// TIA Portal V20 export
TYPE "LBP_typeTMLoad"
TITLE = Tool management / Gestion des outils
// User data type for block LBP_TMLoad [DB71] / Type de données utilisateur pour bloc LBP_TMLoad [DB71]
   STRUCT
      IFNo : Array[1..16] of Bool;   // Interface [number] active / Interface [numéro] active
      Quit : Array[1..16] of Bool;   // Perform Quit-End / Effectuer Quit-End
      TIF : Array[1..16] of Struct
         Loading : Bool;   // Loading the tool / Outil en cours de chargement
         Unloading : Bool;   // Unloading the tool / Outil en cours de déchargement
         Reloading : Bool;   // Relocating the tool / Repositionnement de l'outil
         Positioning : Bool;   // Positioning the magazine / Magasin en cours de positionnement
         PosbyProgram : Bool;   // Initiation by CNC program / Initiation par programme CNC
         PositioningMT : Bool;   // Positioning multitool / Multitool en cours de positionnement
         f0_6 : Bool;   // Reserved / Réservé
         f0_7 : Bool;   // Reserved / Réservé
         PerfStatusError : Bool;   // Negative acknowledge / Acquittement négatif
         n1_1 : Bool;   // Reserved / Réservé
         n1_2 : Bool;   // Reserved / Réservé
         n1_3 : Bool;   // Reserved / Réservé
         n1_4 : Bool;   // Reserved / Réservé
         n1_5 : Bool;   // Reserved / Réservé
         n1_6 : Bool;   // Reserved / Réservé
         DataInDB1071 : Bool;   // Multitool data stored in DB1071 / Données Multitool enregistrées dans DB1071
         Channel : Byte;   // Assigned channel / Canal affecté
         TMNo : Byte;   // Tool management number / Numéro de gestion des outils
         reserved1 : DInt;   // Reserved / Réservé
         reserved2 : DInt;   // Reserved / Réservé
         reserved3 : DInt;   // Reserved / Réservé
         LoadIdent : Int;   // Identification for loading/unloading station / Identifiant de la station de chargement/déchargement
         LoadNo : Int;   // Number of loading station / Numéro de la station de chargement
         SMag : Int;   // Magazine number (source) for unloading/reloading/pos. / Numéro de magasin (source) pour déchargement/rechargement/pos.
         SLoc : Int;   // Location number (source) for unloading/reloading/pos. / Numéro d'emplacement (source) pour déchargement/rechargement/pos.
         TMag : Int;   // Magazine number (target) for loading/reloading / Numéro de magasin (cible) pour déchargement/rechargement
         TLoc : Int;   // Location number (target) for loading/reloading / Numéro d'emplacement (cible) pour déchargement/rechargement
         WithoutMagMoving : Bool;   // HMI Data: without magazine moving / Données HMI : sans déplacement du magasin
         Res2 : Byte;   // Reserved / Réservé
      END_STRUCT;
   END_STRUCT;
   // // TIF[2].Loading : Loading the tool / Outil en cours de chargement
   // // TIF[3].Loading : Loading the tool / Outil en cours de chargement
   // // TIF[4].Loading : Loading the tool / Outil en cours de chargement
   // // TIF[5].Loading : Loading the tool / Outil en cours de chargement
   // // TIF[6].Loading : Loading the tool / Outil en cours de chargement
   // // TIF[7].Loading : Loading the tool / Outil en cours de chargement
   // // TIF[8].Loading : Loading the tool / Outil en cours de chargement
   // // TIF[9].Loading : Loading the tool / Outil en cours de chargement
   // // TIF[10].Loading : Loading the tool / Outil en cours de chargement
   // // TIF[11].Loading : Loading the tool / Outil en cours de chargement
   // // TIF[12].Loading : Loading the tool / Outil en cours de chargement
   // // TIF[13].Loading : Loading the tool / Outil en cours de chargement
   // // TIF[14].Loading : Loading the tool / Outil en cours de chargement
   // // TIF[15].Loading : Loading the tool / Outil en cours de chargement
   // // TIF[16].Loading : Loading the tool / Outil en cours de chargement
   // // TIF[2].Unloading : Unloading the tool / Outil en cours de déchargement
   // // TIF[3].Unloading : Unloading the tool / Outil en cours de déchargement
   // // TIF[4].Unloading : Unloading the tool / Outil en cours de déchargement
   // // TIF[5].Unloading : Unloading the tool / Outil en cours de déchargement
   // // TIF[6].Unloading : Unloading the tool / Outil en cours de déchargement
   // // TIF[7].Unloading : Unloading the tool / Outil en cours de déchargement
   // // TIF[8].Unloading : Unloading the tool / Outil en cours de déchargement
   // // TIF[9].Unloading : Unloading the tool / Outil en cours de déchargement
   // // TIF[10].Unloading : Unloading the tool / Outil en cours de déchargement
   // // TIF[11].Unloading : Unloading the tool / Outil en cours de déchargement
   // // TIF[12].Unloading : Unloading the tool / Outil en cours de déchargement
   // // TIF[13].Unloading : Unloading the tool / Outil en cours de déchargement
   // // TIF[14].Unloading : Unloading the tool / Outil en cours de déchargement
   // // TIF[15].Unloading : Unloading the tool / Outil en cours de déchargement
   // // TIF[16].Unloading : Unloading the tool / Outil en cours de déchargement
   // // TIF[2].Reloading : Relocating the tool / Repositionnement de l'outil
   // // TIF[3].Reloading : Relocating the tool / Repositionnement de l'outil
   // // TIF[4].Reloading : Relocating the tool / Repositionnement de l'outil
   // // TIF[5].Reloading : Relocating the tool / Repositionnement de l'outil
   // // TIF[6].Reloading : Relocating the tool / Repositionnement de l'outil
   // // TIF[7].Reloading : Relocating the tool / Repositionnement de l'outil
   // // TIF[8].Reloading : Relocating the tool / Repositionnement de l'outil
   // // TIF[9].Reloading : Relocating the tool / Repositionnement de l'outil
   // // TIF[10].Reloading : Relocating the tool / Repositionnement de l'outil
   // // TIF[11].Reloading : Relocating the tool / Repositionnement de l'outil
   // // TIF[12].Reloading : Relocating the tool / Repositionnement de l'outil
   // // TIF[13].Reloading : Relocating the tool / Repositionnement de l'outil
   // // TIF[14].Reloading : Relocating the tool / Repositionnement de l'outil
   // // TIF[15].Reloading : Relocating the tool / Repositionnement de l'outil
   // // TIF[16].Reloading : Relocating the tool / Repositionnement de l'outil
   // // TIF[2].Positioning : Positioning the magazine / Magasin en cours de positionnement
   // // TIF[3].Positioning : Positioning the magazine / Magasin en cours de positionnement
   // // TIF[4].Positioning : Positioning the magazine / Magasin en cours de positionnement
   // // TIF[5].Positioning : Positioning the magazine / Magasin en cours de positionnement
   // // TIF[6].Positioning : Positioning the magazine / Magasin en cours de positionnement
   // // TIF[7].Positioning : Positioning the magazine / Magasin en cours de positionnement
   // // TIF[8].Positioning : Positioning the magazine / Magasin en cours de positionnement
   // // TIF[9].Positioning : Positioning the magazine / Magasin en cours de positionnement
   // // TIF[10].Positioning : Positioning the magazine / Magasin en cours de positionnement
   // // TIF[11].Positioning : Positioning the magazine / Magasin en cours de positionnement
   // // TIF[12].Positioning : Positioning the magazine / Magasin en cours de positionnement
   // // TIF[13].Positioning : Positioning the magazine / Magasin en cours de positionnement
   // // TIF[14].Positioning : Positioning the magazine / Magasin en cours de positionnement
   // // TIF[15].Positioning : Positioning the magazine / Magasin en cours de positionnement
   // // TIF[16].Positioning : Positioning the magazine / Magasin en cours de positionnement
   // // TIF[2].PosbyProgram : Initiation by CNC program / Initiation par programme CNC
   // // TIF[3].PosbyProgram : Initiation by CNC program / Initiation par programme CNC
   // // TIF[4].PosbyProgram : Initiation by CNC program / Initiation par programme CNC
   // // TIF[5].PosbyProgram : Initiation by CNC program / Initiation par programme CNC
   // // TIF[6].PosbyProgram : Initiation by CNC program / Initiation par programme CNC
   // // TIF[7].PosbyProgram : Initiation by CNC program / Initiation par programme CNC
   // // TIF[8].PosbyProgram : Initiation by CNC program / Initiation par programme CNC
   // // TIF[9].PosbyProgram : Initiation by CNC program / Initiation par programme CNC
   // // TIF[10].PosbyProgram : Initiation by CNC program / Initiation par programme CNC
   // // TIF[11].PosbyProgram : Initiation by CNC program / Initiation par programme CNC
   // // TIF[12].PosbyProgram : Initiation by CNC program / Initiation par programme CNC
   // // TIF[13].PosbyProgram : Initiation by CNC program / Initiation par programme CNC
   // // TIF[14].PosbyProgram : Initiation by CNC program / Initiation par programme CNC
   // // TIF[15].PosbyProgram : Initiation by CNC program / Initiation par programme CNC
   // // TIF[16].PosbyProgram : Initiation by CNC program / Initiation par programme CNC
   // // TIF[2].PositioningMT : Positioning multitool / Multitool en cours de positionnement
   // // TIF[3].PositioningMT : Positioning multitool / Multitool en cours de positionnement
   // // TIF[4].PositioningMT : Positioning multitool / Multitool en cours de positionnement
   // // TIF[5].PositioningMT : Positioning multitool / Multitool en cours de positionnement
   // // TIF[6].PositioningMT : Positioning multitool / Multitool en cours de positionnement
   // // TIF[7].PositioningMT : Positioning multitool / Multitool en cours de positionnement
   // // TIF[8].PositioningMT : Positioning multitool / Multitool en cours de positionnement
   // // TIF[9].PositioningMT : Positioning multitool / Multitool en cours de positionnement
   // // TIF[10].PositioningMT : Positioning multitool / Multitool en cours de positionnement
   // // TIF[11].PositioningMT : Positioning multitool / Multitool en cours de positionnement
   // // TIF[12].PositioningMT : Positioning multitool / Multitool en cours de positionnement
   // // TIF[13].PositioningMT : Positioning multitool / Multitool en cours de positionnement
   // // TIF[14].PositioningMT : Positioning multitool / Multitool en cours de positionnement
   // // TIF[15].PositioningMT : Positioning multitool / Multitool en cours de positionnement
   // // TIF[16].PositioningMT : Positioning multitool / Multitool en cours de positionnement
   // // TIF[2].f0_6 : Reserved / Réservé
   // // TIF[3].f0_6 : Reserved / Réservé
   // // TIF[4].f0_6 : Reserved / Réservé
   // // TIF[5].f0_6 : Reserved / Réservé
   // // TIF[6].f0_6 : Reserved / Réservé
   // // TIF[7].f0_6 : Reserved / Réservé
   // // TIF[8].f0_6 : Reserved / Réservé
   // // TIF[9].f0_6 : Reserved / Réservé
   // // TIF[10].f0_6 : Reserved / Réservé
   // // TIF[11].f0_6 : Reserved / Réservé
   // // TIF[12].f0_6 : Reserved / Réservé
   // // TIF[13].f0_6 : Reserved / Réservé
   // // TIF[14].f0_6 : Reserved / Réservé
   // // TIF[15].f0_6 : Reserved / Réservé
   // // TIF[16].f0_6 : Reserved / Réservé
   // // TIF[2].f0_7 : Reserved / Réservé
   // // TIF[3].f0_7 : Reserved / Réservé
   // // TIF[4].f0_7 : Reserved / Réservé
   // // TIF[5].f0_7 : Reserved / Réservé
   // // TIF[6].f0_7 : Reserved / Réservé
   // // TIF[7].f0_7 : Reserved / Réservé
   // // TIF[8].f0_7 : Reserved / Réservé
   // // TIF[9].f0_7 : Reserved / Réservé
   // // TIF[10].f0_7 : Reserved / Réservé
   // // TIF[11].f0_7 : Reserved / Réservé
   // // TIF[12].f0_7 : Reserved / Réservé
   // // TIF[13].f0_7 : Reserved / Réservé
   // // TIF[14].f0_7 : Reserved / Réservé
   // // TIF[15].f0_7 : Reserved / Réservé
   // // TIF[16].f0_7 : Reserved / Réservé
   // // TIF[2].PerfStatusError : Negative acknowledge / Acquittement négatif
   // // TIF[3].PerfStatusError : Negative acknowledge / Acquittement négatif
   // // TIF[4].PerfStatusError : Negative acknowledge / Acquittement négatif
   // // TIF[5].PerfStatusError : Negative acknowledge / Acquittement négatif
   // // TIF[6].PerfStatusError : Negative acknowledge / Acquittement négatif
   // // TIF[7].PerfStatusError : Negative acknowledge / Acquittement négatif
   // // TIF[8].PerfStatusError : Negative acknowledge / Acquittement négatif
   // // TIF[9].PerfStatusError : Negative acknowledge / Acquittement négatif
   // // TIF[10].PerfStatusError : Negative acknowledge / Acquittement négatif
   // // TIF[11].PerfStatusError : Negative acknowledge / Acquittement négatif
   // // TIF[12].PerfStatusError : Negative acknowledge / Acquittement négatif
   // // TIF[13].PerfStatusError : Negative acknowledge / Acquittement négatif
   // // TIF[14].PerfStatusError : Negative acknowledge / Acquittement négatif
   // // TIF[15].PerfStatusError : Negative acknowledge / Acquittement négatif
   // // TIF[16].PerfStatusError : Negative acknowledge / Acquittement négatif
   // // TIF[2].n1_1 : Reserved / Réservé
   // // TIF[3].n1_1 : Reserved / Réservé
   // // TIF[4].n1_1 : Reserved / Réservé
   // // TIF[5].n1_1 : Reserved / Réservé
   // // TIF[6].n1_1 : Reserved / Réservé
   // // TIF[7].n1_1 : Reserved / Réservé
   // // TIF[8].n1_1 : Reserved / Réservé
   // // TIF[9].n1_1 : Reserved / Réservé
   // // TIF[10].n1_1 : Reserved / Réservé
   // // TIF[11].n1_1 : Reserved / Réservé
   // // TIF[12].n1_1 : Reserved / Réservé
   // // TIF[13].n1_1 : Reserved / Réservé
   // // TIF[14].n1_1 : Reserved / Réservé
   // // TIF[15].n1_1 : Reserved / Réservé
   // // TIF[16].n1_1 : Reserved / Réservé
   // // TIF[2].n1_2 : Reserved / Réservé
   // // TIF[3].n1_2 : Reserved / Réservé
   // // TIF[4].n1_2 : Reserved / Réservé
   // // TIF[5].n1_2 : Reserved / Réservé
   // // TIF[6].n1_2 : Reserved / Réservé
   // // TIF[7].n1_2 : Reserved / Réservé
   // // TIF[8].n1_2 : Reserved / Réservé
   // // TIF[9].n1_2 : Reserved / Réservé
   // // TIF[10].n1_2 : Reserved / Réservé
   // // TIF[11].n1_2 : Reserved / Réservé
   // // TIF[12].n1_2 : Reserved / Réservé
   // // TIF[13].n1_2 : Reserved / Réservé
   // // TIF[14].n1_2 : Reserved / Réservé
   // // TIF[15].n1_2 : Reserved / Réservé
   // // TIF[16].n1_2 : Reserved / Réservé
   // // TIF[2].n1_3 : Reserved / Réservé
   // // TIF[3].n1_3 : Reserved / Réservé
   // // TIF[4].n1_3 : Reserved / Réservé
   // // TIF[5].n1_3 : Reserved / Réservé
   // // TIF[6].n1_3 : Reserved / Réservé
   // // TIF[7].n1_3 : Reserved / Réservé
   // // TIF[8].n1_3 : Reserved / Réservé
   // // TIF[9].n1_3 : Reserved / Réservé
   // // TIF[10].n1_3 : Reserved / Réservé
   // // TIF[11].n1_3 : Reserved / Réservé
   // // TIF[12].n1_3 : Reserved / Réservé
   // // TIF[13].n1_3 : Reserved / Réservé
   // // TIF[14].n1_3 : Reserved / Réservé
   // // TIF[15].n1_3 : Reserved / Réservé
   // // TIF[16].n1_3 : Reserved / Réservé
   // // TIF[2].n1_4 : Reserved / Réservé
   // // TIF[3].n1_4 : Reserved / Réservé
   // // TIF[4].n1_4 : Reserved / Réservé
   // // TIF[5].n1_4 : Reserved / Réservé
   // // TIF[6].n1_4 : Reserved / Réservé
   // // TIF[7].n1_4 : Reserved / Réservé
   // // TIF[8].n1_4 : Reserved / Réservé
   // // TIF[9].n1_4 : Reserved / Réservé
   // // TIF[10].n1_4 : Reserved / Réservé
   // // TIF[11].n1_4 : Reserved / Réservé
   // // TIF[12].n1_4 : Reserved / Réservé
   // // TIF[13].n1_4 : Reserved / Réservé
   // // TIF[14].n1_4 : Reserved / Réservé
   // // TIF[15].n1_4 : Reserved / Réservé
   // // TIF[16].n1_4 : Reserved / Réservé
   // // TIF[2].n1_5 : Reserved / Réservé
   // // TIF[3].n1_5 : Reserved / Réservé
   // // TIF[4].n1_5 : Reserved / Réservé
   // // TIF[5].n1_5 : Reserved / Réservé
   // // TIF[6].n1_5 : Reserved / Réservé
   // // TIF[7].n1_5 : Reserved / Réservé
   // // TIF[8].n1_5 : Reserved / Réservé
   // // TIF[9].n1_5 : Reserved / Réservé
   // // TIF[10].n1_5 : Reserved / Réservé
   // // TIF[11].n1_5 : Reserved / Réservé
   // // TIF[12].n1_5 : Reserved / Réservé
   // // TIF[13].n1_5 : Reserved / Réservé
   // // TIF[14].n1_5 : Reserved / Réservé
   // // TIF[15].n1_5 : Reserved / Réservé
   // // TIF[16].n1_5 : Reserved / Réservé
   // // TIF[2].n1_6 : Reserved / Réservé
   // // TIF[3].n1_6 : Reserved / Réservé
   // // TIF[4].n1_6 : Reserved / Réservé
   // // TIF[5].n1_6 : Reserved / Réservé
   // // TIF[6].n1_6 : Reserved / Réservé
   // // TIF[7].n1_6 : Reserved / Réservé
   // // TIF[8].n1_6 : Reserved / Réservé
   // // TIF[9].n1_6 : Reserved / Réservé
   // // TIF[10].n1_6 : Reserved / Réservé
   // // TIF[11].n1_6 : Reserved / Réservé
   // // TIF[12].n1_6 : Reserved / Réservé
   // // TIF[13].n1_6 : Reserved / Réservé
   // // TIF[14].n1_6 : Reserved / Réservé
   // // TIF[15].n1_6 : Reserved / Réservé
   // // TIF[16].n1_6 : Reserved / Réservé
   // // TIF[2].DataInDB1071 : Multitool data stored in DB1071 / Données Multitool enregistrées dans DB1071
   // // TIF[3].DataInDB1071 : Multitool data stored in DB1071 / Données Multitool enregistrées dans DB1071
   // // TIF[4].DataInDB1071 : Multitool data stored in DB1071 / Données Multitool enregistrées dans DB1071
   // // TIF[5].DataInDB1071 : Multitool data stored in DB1071 / Données Multitool enregistrées dans DB1071
   // // TIF[6].DataInDB1071 : Multitool data stored in DB1071 / Données Multitool enregistrées dans DB1071
   // // TIF[7].DataInDB1071 : Multitool data stored in DB1071 / Données Multitool enregistrées dans DB1071
   // // TIF[8].DataInDB1071 : Multitool data stored in DB1071 / Données Multitool enregistrées dans DB1071
   // // TIF[9].DataInDB1071 : Multitool data stored in DB1071 / Données Multitool enregistrées dans DB1071
   // // TIF[10].DataInDB1071 : Multitool data stored in DB1071 / Données Multitool enregistrées dans DB1071
   // // TIF[11].DataInDB1071 : Multitool data stored in DB1071 / Données Multitool enregistrées dans DB1071
   // // TIF[12].DataInDB1071 : Multitool data stored in DB1071 / Données Multitool enregistrées dans DB1071
   // // TIF[13].DataInDB1071 : Multitool data stored in DB1071 / Données Multitool enregistrées dans DB1071
   // // TIF[14].DataInDB1071 : Multitool data stored in DB1071 / Données Multitool enregistrées dans DB1071
   // // TIF[15].DataInDB1071 : Multitool data stored in DB1071 / Données Multitool enregistrées dans DB1071
   // // TIF[16].DataInDB1071 : Multitool data stored in DB1071 / Données Multitool enregistrées dans DB1071
   // // TIF[2].Channel : Assigned channel / Canal affecté
   // // TIF[3].Channel : Assigned channel / Canal affecté
   // // TIF[4].Channel : Assigned channel / Canal affecté
   // // TIF[5].Channel : Assigned channel / Canal affecté
   // // TIF[6].Channel : Assigned channel / Canal affecté
   // // TIF[7].Channel : Assigned channel / Canal affecté
   // // TIF[8].Channel : Assigned channel / Canal affecté
   // // TIF[9].Channel : Assigned channel / Canal affecté
   // // TIF[10].Channel : Assigned channel / Canal affecté
   // // TIF[11].Channel : Assigned channel / Canal affecté
   // // TIF[12].Channel : Assigned channel / Canal affecté
   // // TIF[13].Channel : Assigned channel / Canal affecté
   // // TIF[14].Channel : Assigned channel / Canal affecté
   // // TIF[15].Channel : Assigned channel / Canal affecté
   // // TIF[16].Channel : Assigned channel / Canal affecté
   // // TIF[2].TMNo : Tool management number / Numéro de gestion des outils
   // // TIF[3].TMNo : Tool management number / Numéro de gestion des outils
   // // TIF[4].TMNo : Tool management number / Numéro de gestion des outils
   // // TIF[5].TMNo : Tool management number / Numéro de gestion des outils
   // // TIF[6].TMNo : Tool management number / Numéro de gestion des outils
   // // TIF[7].TMNo : Tool management number / Numéro de gestion des outils
   // // TIF[8].TMNo : Tool management number / Numéro de gestion des outils
   // // TIF[9].TMNo : Tool management number / Numéro de gestion des outils
   // // TIF[10].TMNo : Tool management number / Numéro de gestion des outils
   // // TIF[11].TMNo : Tool management number / Numéro de gestion des outils
   // // TIF[12].TMNo : Tool management number / Numéro de gestion des outils
   // // TIF[13].TMNo : Tool management number / Numéro de gestion des outils
   // // TIF[14].TMNo : Tool management number / Numéro de gestion des outils
   // // TIF[15].TMNo : Tool management number / Numéro de gestion des outils
   // // TIF[16].TMNo : Tool management number / Numéro de gestion des outils
   // // TIF[2].reserved1 : Reserved / Réservé
   // // TIF[3].reserved1 : Reserved / Réservé
   // // TIF[4].reserved1 : Reserved / Réservé
   // // TIF[5].reserved1 : Reserved / Réservé
   // // TIF[6].reserved1 : Reserved / Réservé
   // // TIF[7].reserved1 : Reserved / Réservé
   // // TIF[8].reserved1 : Reserved / Réservé
   // // TIF[9].reserved1 : Reserved / Réservé
   // // TIF[10].reserved1 : Reserved / Réservé
   // // TIF[11].reserved1 : Reserved / Réservé
   // // TIF[12].reserved1 : Reserved / Réservé
   // // TIF[13].reserved1 : Reserved / Réservé
   // // TIF[14].reserved1 : Reserved / Réservé
   // // TIF[15].reserved1 : Reserved / Réservé
   // // TIF[16].reserved1 : Reserved / Réservé
   // // TIF[2].reserved2 : Reserved / Réservé
   // // TIF[3].reserved2 : Reserved / Réservé
   // // TIF[4].reserved2 : Reserved / Réservé
   // // TIF[5].reserved2 : Reserved / Réservé
   // // TIF[6].reserved2 : Reserved / Réservé
   // // TIF[7].reserved2 : Reserved / Réservé
   // // TIF[8].reserved2 : Reserved / Réservé
   // // TIF[9].reserved2 : Reserved / Réservé
   // // TIF[10].reserved2 : Reserved / Réservé
   // // TIF[11].reserved2 : Reserved / Réservé
   // // TIF[12].reserved2 : Reserved / Réservé
   // // TIF[13].reserved2 : Reserved / Réservé
   // // TIF[14].reserved2 : Reserved / Réservé
   // // TIF[15].reserved2 : Reserved / Réservé
   // // TIF[16].reserved2 : Reserved / Réservé
   // // TIF[2].reserved3 : Reserved / Réservé
   // // TIF[3].reserved3 : Reserved / Réservé
   // // TIF[4].reserved3 : Reserved / Réservé
   // // TIF[5].reserved3 : Reserved / Réservé
   // // TIF[6].reserved3 : Reserved / Réservé
   // // TIF[7].reserved3 : Reserved / Réservé
   // // TIF[8].reserved3 : Reserved / Réservé
   // // TIF[9].reserved3 : Reserved / Réservé
   // // TIF[10].reserved3 : Reserved / Réservé
   // // TIF[11].reserved3 : Reserved / Réservé
   // // TIF[12].reserved3 : Reserved / Réservé
   // // TIF[13].reserved3 : Reserved / Réservé
   // // TIF[14].reserved3 : Reserved / Réservé
   // // TIF[15].reserved3 : Reserved / Réservé
   // // TIF[16].reserved3 : Reserved / Réservé
   // // TIF[2].LoadIdent : Identification for loading/unloading station / Identifiant de la station de chargement/déchargement
   // // TIF[3].LoadIdent : Identification for loading/unloading station / Identifiant de la station de chargement/déchargement
   // // TIF[4].LoadIdent : Identification for loading/unloading station / Identifiant de la station de chargement/déchargement
   // // TIF[5].LoadIdent : Identification for loading/unloading station / Identifiant de la station de chargement/déchargement
   // // TIF[6].LoadIdent : Identification for loading/unloading station / Identifiant de la station de chargement/déchargement
   // // TIF[7].LoadIdent : Identification for loading/unloading station / Identifiant de la station de chargement/déchargement
   // // TIF[8].LoadIdent : Identification for loading/unloading station / Identifiant de la station de chargement/déchargement
   // // TIF[9].LoadIdent : Identification for loading/unloading station / Identifiant de la station de chargement/déchargement
   // // TIF[10].LoadIdent : Identification for loading/unloading station / Identifiant de la station de chargement/déchargement
   // // TIF[11].LoadIdent : Identification for loading/unloading station / Identifiant de la station de chargement/déchargement
   // // TIF[12].LoadIdent : Identification for loading/unloading station / Identifiant de la station de chargement/déchargement
   // // TIF[13].LoadIdent : Identification for loading/unloading station / Identifiant de la station de chargement/déchargement
   // // TIF[14].LoadIdent : Identification for loading/unloading station / Identifiant de la station de chargement/déchargement
   // // TIF[15].LoadIdent : Identification for loading/unloading station / Identifiant de la station de chargement/déchargement
   // // TIF[16].LoadIdent : Identification for loading/unloading station / Identifiant de la station de chargement/déchargement
   // // TIF[2].LoadNo : Number of loading station / Numéro de la station de chargement
   // // TIF[3].LoadNo : Number of loading station / Numéro de la station de chargement
   // // TIF[4].LoadNo : Number of loading station / Numéro de la station de chargement
   // // TIF[5].LoadNo : Number of loading station / Numéro de la station de chargement
   // // TIF[6].LoadNo : Number of loading station / Numéro de la station de chargement
   // // TIF[7].LoadNo : Number of loading station / Numéro de la station de chargement
   // // TIF[8].LoadNo : Number of loading station / Numéro de la station de chargement
   // // TIF[9].LoadNo : Number of loading station / Numéro de la station de chargement
   // // TIF[10].LoadNo : Number of loading station / Numéro de la station de chargement
   // // TIF[11].LoadNo : Number of loading station / Numéro de la station de chargement
   // // TIF[12].LoadNo : Number of loading station / Numéro de la station de chargement
   // // TIF[13].LoadNo : Number of loading station / Numéro de la station de chargement
   // // TIF[14].LoadNo : Number of loading station / Numéro de la station de chargement
   // // TIF[15].LoadNo : Number of loading station / Numéro de la station de chargement
   // // TIF[16].LoadNo : Number of loading station / Numéro de la station de chargement
   // // TIF[2].SMag : Magazine number (source) for unloading/reloading/pos. / Numéro de magasin (source) pour déchargement/rechargement/pos.
   // // TIF[3].SMag : Magazine number (source) for unloading/reloading/pos. / Numéro de magasin (source) pour déchargement/rechargement/pos.
   // // TIF[4].SMag : Magazine number (source) for unloading/reloading/pos. / Numéro de magasin (source) pour déchargement/rechargement/pos.
   // // TIF[5].SMag : Magazine number (source) for unloading/reloading/pos. / Numéro de magasin (source) pour déchargement/rechargement/pos.
   // // TIF[6].SMag : Magazine number (source) for unloading/reloading/pos. / Numéro de magasin (source) pour déchargement/rechargement/pos.
   // // TIF[7].SMag : Magazine number (source) for unloading/reloading/pos. / Numéro de magasin (source) pour déchargement/rechargement/pos.
   // // TIF[8].SMag : Magazine number (source) for unloading/reloading/pos. / Numéro de magasin (source) pour déchargement/rechargement/pos.
   // // TIF[9].SMag : Magazine number (source) for unloading/reloading/pos. / Numéro de magasin (source) pour déchargement/rechargement/pos.
   // // TIF[10].SMag : Magazine number (source) for unloading/reloading/pos. / Numéro de magasin (source) pour déchargement/rechargement/pos.
   // // TIF[11].SMag : Magazine number (source) for unloading/reloading/pos. / Numéro de magasin (source) pour déchargement/rechargement/pos.
   // // TIF[12].SMag : Magazine number (source) for unloading/reloading/pos. / Numéro de magasin (source) pour déchargement/rechargement/pos.
   // // TIF[13].SMag : Magazine number (source) for unloading/reloading/pos. / Numéro de magasin (source) pour déchargement/rechargement/pos.
   // // TIF[14].SMag : Magazine number (source) for unloading/reloading/pos. / Numéro de magasin (source) pour déchargement/rechargement/pos.
   // // TIF[15].SMag : Magazine number (source) for unloading/reloading/pos. / Numéro de magasin (source) pour déchargement/rechargement/pos.
   // // TIF[16].SMag : Magazine number (source) for unloading/reloading/pos. / Numéro de magasin (source) pour déchargement/rechargement/pos.
   // // TIF[2].SLoc : Location number (source) for unloading/reloading/pos. / Numéro d'emplacement (source) pour déchargement/rechargement/pos.
   // // TIF[3].SLoc : Location number (source) for unloading/reloading/pos. / Numéro d'emplacement (source) pour déchargement/rechargement/pos.
   // // TIF[4].SLoc : Location number (source) for unloading/reloading/pos. / Numéro d'emplacement (source) pour déchargement/rechargement/pos.
   // // TIF[5].SLoc : Location number (source) for unloading/reloading/pos. / Numéro d'emplacement (source) pour déchargement/rechargement/pos.
   // // TIF[6].SLoc : Location number (source) for unloading/reloading/pos. / Numéro d'emplacement (source) pour déchargement/rechargement/pos.
   // // TIF[7].SLoc : Location number (source) for unloading/reloading/pos. / Numéro d'emplacement (source) pour déchargement/rechargement/pos.
   // // TIF[8].SLoc : Location number (source) for unloading/reloading/pos. / Numéro d'emplacement (source) pour déchargement/rechargement/pos.
   // // TIF[9].SLoc : Location number (source) for unloading/reloading/pos. / Numéro d'emplacement (source) pour déchargement/rechargement/pos.
   // // TIF[10].SLoc : Location number (source) for unloading/reloading/pos. / Numéro d'emplacement (source) pour déchargement/rechargement/pos.
   // // TIF[11].SLoc : Location number (source) for unloading/reloading/pos. / Numéro d'emplacement (source) pour déchargement/rechargement/pos.
   // // TIF[12].SLoc : Location number (source) for unloading/reloading/pos. / Numéro d'emplacement (source) pour déchargement/rechargement/pos.
   // // TIF[13].SLoc : Location number (source) for unloading/reloading/pos. / Numéro d'emplacement (source) pour déchargement/rechargement/pos.
   // // TIF[14].SLoc : Location number (source) for unloading/reloading/pos. / Numéro d'emplacement (source) pour déchargement/rechargement/pos.
   // // TIF[15].SLoc : Location number (source) for unloading/reloading/pos. / Numéro d'emplacement (source) pour déchargement/rechargement/pos.
   // // TIF[16].SLoc : Location number (source) for unloading/reloading/pos. / Numéro d'emplacement (source) pour déchargement/rechargement/pos.
   // // TIF[2].TMag : Magazine number (target) for loading/reloading / Numéro de magasin (cible) pour déchargement/rechargement
   // // TIF[3].TMag : Magazine number (target) for loading/reloading / Numéro de magasin (cible) pour déchargement/rechargement
   // // TIF[4].TMag : Magazine number (target) for loading/reloading / Numéro de magasin (cible) pour déchargement/rechargement
   // // TIF[5].TMag : Magazine number (target) for loading/reloading / Numéro de magasin (cible) pour déchargement/rechargement
   // // TIF[6].TMag : Magazine number (target) for loading/reloading / Numéro de magasin (cible) pour déchargement/rechargement
   // // TIF[7].TMag : Magazine number (target) for loading/reloading / Numéro de magasin (cible) pour déchargement/rechargement
   // // TIF[8].TMag : Magazine number (target) for loading/reloading / Numéro de magasin (cible) pour déchargement/rechargement
   // // TIF[9].TMag : Magazine number (target) for loading/reloading / Numéro de magasin (cible) pour déchargement/rechargement
   // // TIF[10].TMag : Magazine number (target) for loading/reloading / Numéro de magasin (cible) pour déchargement/rechargement
   // // TIF[11].TMag : Magazine number (target) for loading/reloading / Numéro de magasin (cible) pour déchargement/rechargement
   // // TIF[12].TMag : Magazine number (target) for loading/reloading / Numéro de magasin (cible) pour déchargement/rechargement
   // // TIF[13].TMag : Magazine number (target) for loading/reloading / Numéro de magasin (cible) pour déchargement/rechargement
   // // TIF[14].TMag : Magazine number (target) for loading/reloading / Numéro de magasin (cible) pour déchargement/rechargement
   // // TIF[15].TMag : Magazine number (target) for loading/reloading / Numéro de magasin (cible) pour déchargement/rechargement
   // // TIF[16].TMag : Magazine number (target) for loading/reloading / Numéro de magasin (cible) pour déchargement/rechargement
   // // TIF[2].TLoc : Location number (target) for loading/reloading / Numéro d'emplacement (cible) pour déchargement/rechargement
   // // TIF[3].TLoc : Location number (target) for loading/reloading / Numéro d'emplacement (cible) pour déchargement/rechargement
   // // TIF[4].TLoc : Location number (target) for loading/reloading / Numéro d'emplacement (cible) pour déchargement/rechargement
   // // TIF[5].TLoc : Location number (target) for loading/reloading / Numéro d'emplacement (cible) pour déchargement/rechargement
   // // TIF[6].TLoc : Location number (target) for loading/reloading / Numéro d'emplacement (cible) pour déchargement/rechargement
   // // TIF[7].TLoc : Location number (target) for loading/reloading / Numéro d'emplacement (cible) pour déchargement/rechargement
   // // TIF[8].TLoc : Location number (target) for loading/reloading / Numéro d'emplacement (cible) pour déchargement/rechargement
   // // TIF[9].TLoc : Location number (target) for loading/reloading / Numéro d'emplacement (cible) pour déchargement/rechargement
   // // TIF[10].TLoc : Location number (target) for loading/reloading / Numéro d'emplacement (cible) pour déchargement/rechargement
   // // TIF[11].TLoc : Location number (target) for loading/reloading / Numéro d'emplacement (cible) pour déchargement/rechargement
   // // TIF[12].TLoc : Location number (target) for loading/reloading / Numéro d'emplacement (cible) pour déchargement/rechargement
   // // TIF[13].TLoc : Location number (target) for loading/reloading / Numéro d'emplacement (cible) pour déchargement/rechargement
   // // TIF[14].TLoc : Location number (target) for loading/reloading / Numéro d'emplacement (cible) pour déchargement/rechargement
   // // TIF[15].TLoc : Location number (target) for loading/reloading / Numéro d'emplacement (cible) pour déchargement/rechargement
   // // TIF[16].TLoc : Location number (target) for loading/reloading / Numéro d'emplacement (cible) pour déchargement/rechargement
   // // TIF[2].WithoutMagMoving : HMI Data: without magazine moving / Données HMI : sans déplacement du magasin
   // // TIF[3].WithoutMagMoving : HMI Data: without magazine moving / Données HMI : sans déplacement du magasin
   // // TIF[4].WithoutMagMoving : HMI Data: without magazine moving / Données HMI : sans déplacement du magasin
   // // TIF[5].WithoutMagMoving : HMI Data: without magazine moving / Données HMI : sans déplacement du magasin
   // // TIF[6].WithoutMagMoving : HMI Data: without magazine moving / Données HMI : sans déplacement du magasin
   // // TIF[7].WithoutMagMoving : HMI Data: without magazine moving / Données HMI : sans déplacement du magasin
   // // TIF[8].WithoutMagMoving : HMI Data: without magazine moving / Données HMI : sans déplacement du magasin
   // // TIF[9].WithoutMagMoving : HMI Data: without magazine moving / Données HMI : sans déplacement du magasin
   // // TIF[10].WithoutMagMoving : HMI Data: without magazine moving / Données HMI : sans déplacement du magasin
   // // TIF[11].WithoutMagMoving : HMI Data: without magazine moving / Données HMI : sans déplacement du magasin
   // // TIF[12].WithoutMagMoving : HMI Data: without magazine moving / Données HMI : sans déplacement du magasin
   // // TIF[13].WithoutMagMoving : HMI Data: without magazine moving / Données HMI : sans déplacement du magasin
   // // TIF[14].WithoutMagMoving : HMI Data: without magazine moving / Données HMI : sans déplacement du magasin
   // // TIF[15].WithoutMagMoving : HMI Data: without magazine moving / Données HMI : sans déplacement du magasin
   // // TIF[16].WithoutMagMoving : HMI Data: without magazine moving / Données HMI : sans déplacement du magasin
   // // TIF[2].Res2 : Reserved / Réservé
   // // TIF[3].Res2 : Reserved / Réservé
   // // TIF[4].Res2 : Reserved / Réservé
   // // TIF[5].Res2 : Reserved / Réservé
   // // TIF[6].Res2 : Reserved / Réservé
   // // TIF[7].Res2 : Reserved / Réservé
   // // TIF[8].Res2 : Reserved / Réservé
   // // TIF[9].Res2 : Reserved / Réservé
   // // TIF[10].Res2 : Reserved / Réservé
   // // TIF[11].Res2 : Reserved / Réservé
   // // TIF[12].Res2 : Reserved / Réservé
   // // TIF[13].Res2 : Reserved / Réservé
   // // TIF[14].Res2 : Reserved / Réservé
   // // TIF[15].Res2 : Reserved / Réservé
   // // TIF[16].Res2 : Reserved / Réservé
END_TYPE
